// TIA Portal V18 export
DATA_BLOCK "Refilling"   // DB136
{ S7_Optimized_Access := 'TRUE' }
VERSION : 0.1
// stored: AutoNumber true, DBAccessibleFromOPCUA true, IsOnlyStoredInLoadMemory false, IsRetainMemResEnabled false, IsWriteProtectedInAS false, MemoryReserve 100
   VAR
      Running : Struct
         A1 : Bool;
         A2 : Bool;
         B1 : Bool;
      END_STRUCT;
      "Control A1" : Struct
         "Start Refilling" : Bool;
         "refilling failed" : Bool;
      END_STRUCT;
      "Control A2" : Struct
         "Start Refilling" : Bool;
         "refilling failed" : Bool;
      END_STRUCT;
      "Control B1" : Struct
         "Start Refilling" : Bool;
         "refilling failed" : Bool;
      END_STRUCT;
      "Output A1" : Struct
         "Run vacuum PUMP" : Bool;
         "Open Vaccum Valve" : Bool;
         "Open refilling Valve" : Bool;
         "Pump minimum run time okay" : Bool;
      END_STRUCT;
      "Output A2" : Struct
         "Run vacuum PUMP" : Bool;
         "Open Vaccum Valve" : Bool;
         "Open refilling Valve" : Bool;
         "Pump minimum run time okay" : Bool;
      END_STRUCT;
      "Output B1" : Struct
         "Run vacuum PUMP" : Bool;
         "Open Vaccum Valve" : Bool;
         "Open refilling Valve" : Bool;
         "Pump minimum run time okay" : Bool;
      END_STRUCT;
      "filling level A1" : Struct
         "Filling level reached" : Bool;
         "Filling failed" : Bool;
         "Previous value" : Real;
         "current value" : Real;
         "start Compare" : Bool;
         "stop compare" : Bool;
      END_STRUCT;
      "filling level A2" : Struct
         "Filling level reached" : Bool;
         "Filling failed" : Bool;
         "Previous value" : Real;
         "current value" : Real;
         "start Compare" : Bool;
         "stop compare" : Bool;
      END_STRUCT;
      "filling level B1" : Struct
         "Filling level reached" : Bool;
         "Filling failed" : Bool;
         "Previous value" : Real;
         "current value" : Real;
         "start Compare" : Bool;
         "stop compare" : Bool;
      END_STRUCT;
   END_VAR
   VAR RETAIN
      "level increase in 30s" : Struct
         "A" : Real;
         "B" : Real;
      END_STRUCT;
      PressureExaustTime : DInt;
   END_VAR
   VAR
      PressureReleaseA : Bool;
      PressureReleaseB : Bool;
      "Start Auto Refill A" : Bool;
      "Start Auto Refill B" : Bool;
   END_VAR
   VAR RETAIN
      PressureExaustTimeS : DInt;
   END_VAR
   VAR
      Temp1 : Bool;
      Temp2 : Bool;
   END_VAR
BEGIN
END_DATA_BLOCK
